{attribute 'TcGenerated'}
{attribute 'no-analysis'}
{attribute 'linkalways'}
// This function has been automatically generated from the project information.
VAR_GLOBAL CONSTANT
	{attribute 'const_non_replaced'}
	stLibVersion_TcTcpUdpRT : ST_LibVersion := (iMajor := 1, iMinor := 0, iBuild := 0, iRevision := 1, nFlags := 0, sVersion := '1.0.0.1');
END_VAR

(* stored: Version 1.1.0.1
   GVL Global_Version: Id {ae8fcb2e-4429-094b-2e1c-47b6d70b42a3} *)
